INTERFACE I_SynchronousRpcHandlers

PROPERTY PUBLIC HasHandlers : BOOL
GET
END_GET
END_PROPERTY

METHOD PUBLIC TryGetByMethodName : BOOL
VAR_INPUT
	MethodName : T_MAXSTRING;
	Destination : REFERENCE TO I_SynchronousRpcHandler;
END_VAR
END_METHOD

END_INTERFACE

(* stored: Version 1.1.0.1, ProductVersion 3.1.4024.12
   Itf I_SynchronousRpcHandlers: Id {80025cfc-f7e6-0fd1-30c9-e00b0ba7ba6b}
   Property HasHandlers: Id {fa1fa595-533d-43ca-86a0-1cfbd9cf2b27}
   Get Get: Id {c74cf47c-051a-480c-91dd-36c0a377744f}
   Method TryGetByMethodName: Id {be929ac2-bf47-0767-3f83-858d5787a6e3} *)
